// TIA Portal V18 export
// export: Created 2025-12-01T17:50:52.6792263Z, ExportSetting None, DisplayName Totally Integrated Automation Portal, DisplayVersion V18 Update 5, DisplayName TIA Portal Openness, DisplayVersion V18 Update 5, DisplayName TIA Portal Teamcenter Gateway, DisplayVersion V18, DisplayName TIA Portal Version Control Interface, DisplayVersion V18, DisplayName STEP 7 Professional, DisplayVersion V18 Update 5, DisplayName STEP 7 Safety, DisplayVersion V18, DisplayName WinCC Professional, DisplayVersion V18 Update 5
FUNCTION_BLOCK "ST10_Flow23_KReserveLifting"   // FB1093, GRAPH
// stored: AcknowledgeErrorsRequired false, AutoNumber false, GraphVersion 6.0, InitialValuesAcquisition false, SetENOAutomatically false
   // inherited from GRAPH_BASE
   VAR_INPUT
      iSysInface : "RCS_SysComInterface_V1";
   END_VAR
   VAR_IN_OUT
      ioPM_Inface : "RCS_PMInterface_V1";
      ioStatus : Int;
   END_VAR
   VAR
      sCtrlMode { S7_SetPoint := 'True'} : "SysFlowCtrlGraph";
      sUpdMES_Data : Bool;   // 更新MES数据
      工件放行中 : Bool;
      前站站号 { ExternalAccessible := 'False'; ExternalVisible := 'False'; ExternalWritable := 'False'} : UInt;
      本站站号 { ExternalAccessible := 'False'; ExternalVisible := 'False'; ExternalWritable := 'False'} : UInt;
      弹窗Temp : Array[1..10] of Int;
      AlarmID : Int;
      TON { S7_SetPoint := 'True'} : Array[0..10] of TON_TIME;
      TOF { S7_SetPoint := 'True'} : Array[0..10] of TOF_TIME;
      sUP { S7_SetPoint := 'True'} : Array[0..10] of Bool;
      更新RFID完成 : Bool;
   END_VAR
   VAR_TEMP
      Tempresult : USInt;
      本站站号乘10 : UInt;
   END_VAR
   // // TON[0] : 托盘流入1托盘到位传感器 / iA-Rotating product Check
   // // TON[1] : 托盘流入1托盘到位传感器
   // // TON[2] : 托盘流入1产品有无传感器
   // // TON[3] : 托盘流入1产品有无传感器
   // // TON[4] : 托盘流入1姿态检测光电2
   // // TON[5] : 托盘流入1姿态检测光电3
   // // TON[0].Q : 托盘流入1托盘到位 / iA-Rotating product Check
   // // TON[1].Q : 托盘流入1托盘无
   // // TON[2].Q : 托盘流入1有产品
   // // TON[3].Q : 托盘流入1无产品
   // // TON[4].Q : 托盘流入1姿态检测光电2
   // // TON[5].Q : 托盘流入1姿态检测光电3
   // // TOF[1] : iA-Rotating product Check
BEGIN
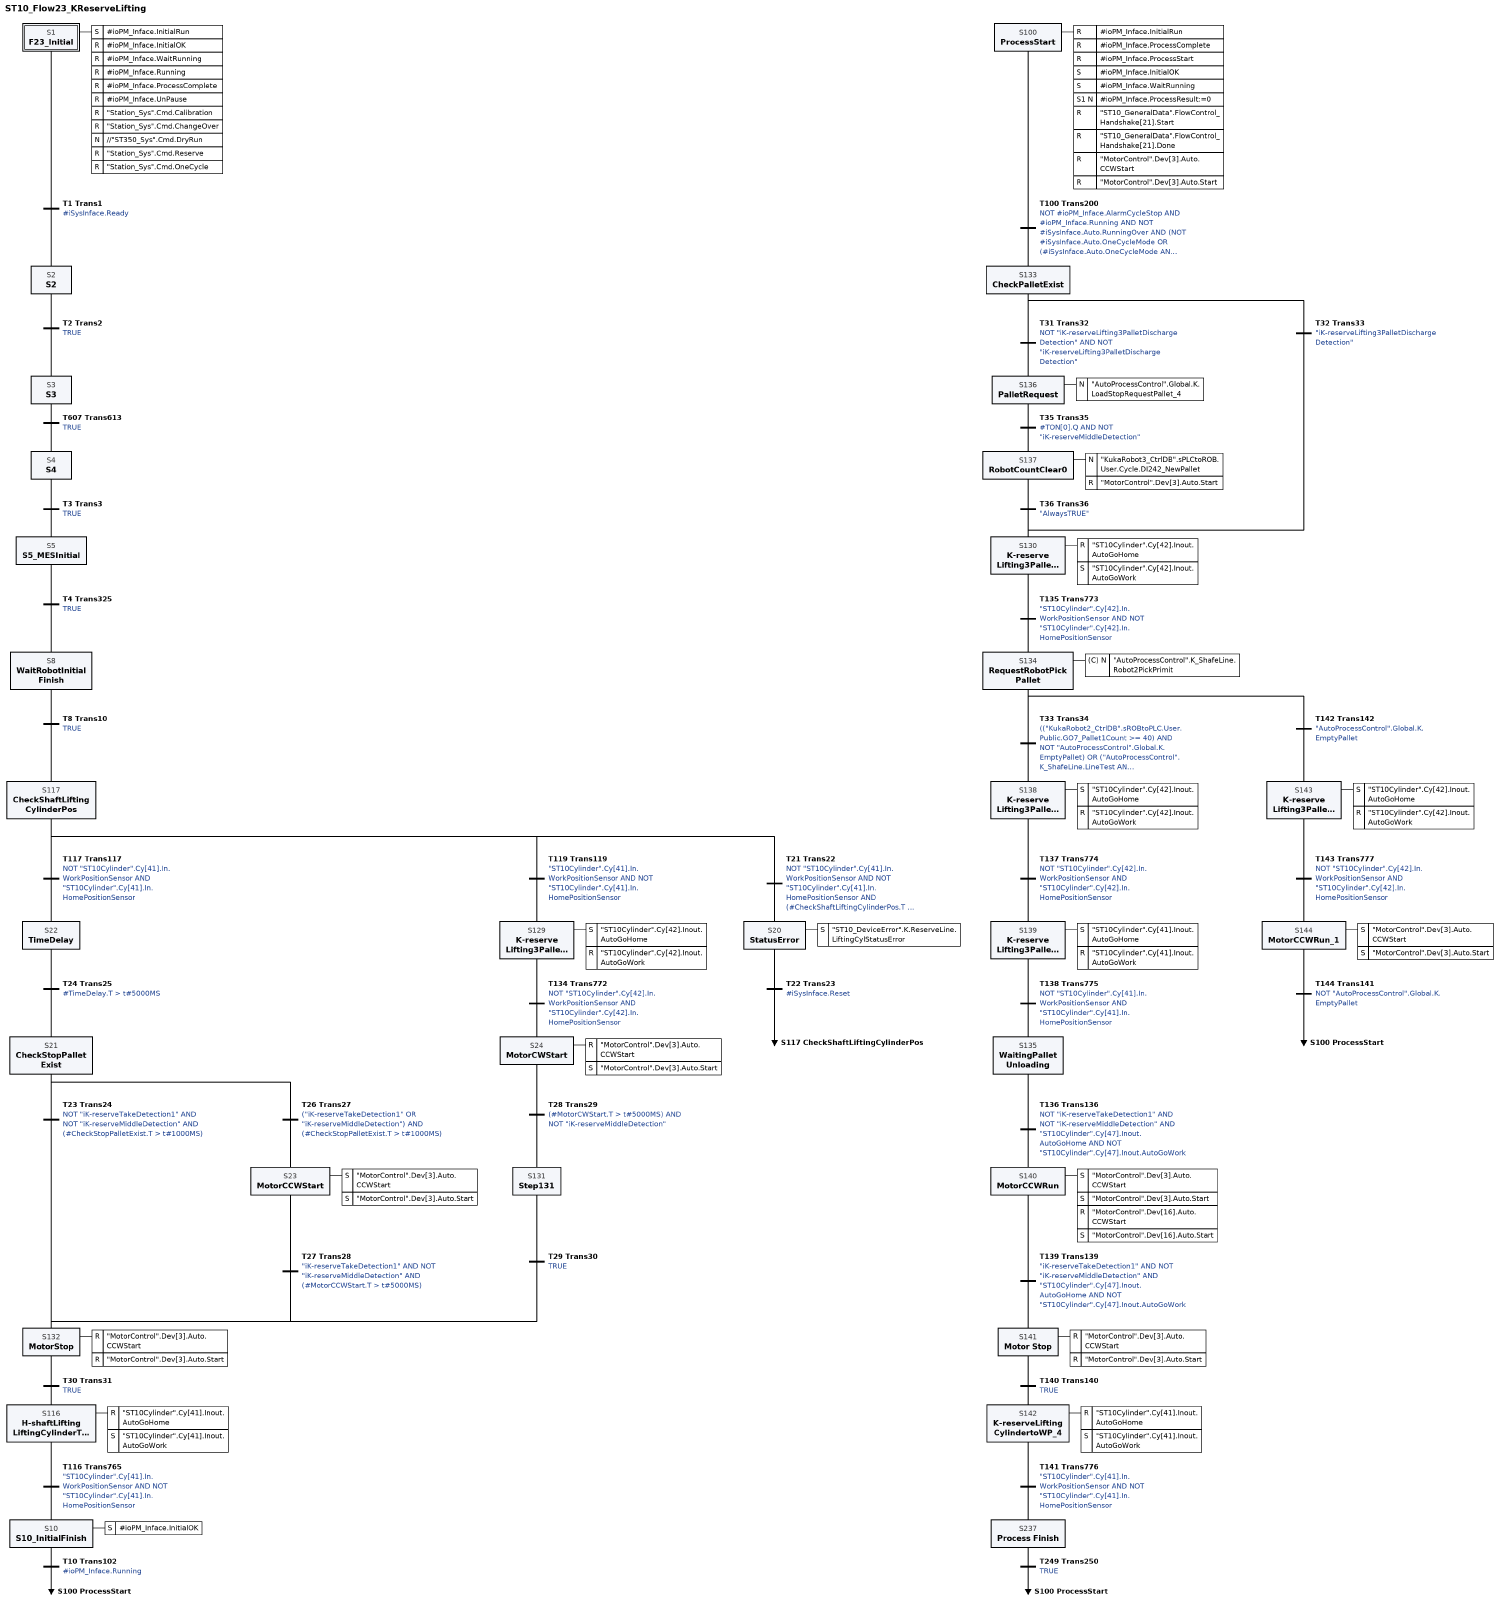
   // permanent pre-instructions
   NETWORK 1
      #TON[10].TON(IN := "AlwaysTRUE" AND "Station_Sys".Alarm.ImmediatelyStop, PT := T#300ms);
      #ioPM_Inface.AlarmImdilyStop := #TON[10].Q;
      #ioPM_Inface.AlarmCycleStop := "AlwaysTRUE" AND "Station_Sys".Alarm.CycleStop;
   NETWORK 2
      IF NOT False THEN
          #sCtrlMode(iSysInface := #iSysInface, ioPM_Inface := #ioPM_Inface, ioGraphCtrl := #RT_DATA.MOP);   // "SysFlowCtrlGraph"
      END_IF;
   NETWORK 3
      #TON[0].TON(IN := "AlwaysTRUE" AND "iK-reserveLifting3PalletDischargeDetection", PT := t#1000ms);   // 工位11有托盘
      #TOF[1].TOF(IN := "AlwaysTRUE" AND NOT "iK-reserveLifting3PalletDischargeDetection", PT := T#300ms);   // 工位无托盘
      #TON[2].TON(IN := "AlwaysTRUE", PT := T#300ms);
      #TOF[3].TOF(IN := "AlwaysTRUE", PT := T#300ms);
      #TON[4].TON(IN := "AlwaysTRUE", PT := T#300ms);
      #TOF[5].TOF(IN := "AlwaysTRUE", PT := T#300ms);
   NETWORK 4
      #前站站号 := 345;
      #本站站号 := 350;

   // sequencer 1: S01-S99 初始化 / S01-S99 Initial
   INITIAL_STEP F23_Initial:   // S1, max time T#10S, warning time T#7S
              S    #ioPM_Inface.InitialRun
              R    #ioPM_Inface.InitialOK
              R    #ioPM_Inface.WaitRunning
              R    #ioPM_Inface.Running
              R    #ioPM_Inface.ProcessComplete
              R    #ioPM_Inface.UnPause
              R    "Station_Sys".Cmd.Calibration
              R    "Station_Sys".Cmd.ChangeOver
                   //"ST350_Sys".Cmd.DryRun
              R    "Station_Sys".Cmd.Reserve
              R    "Station_Sys".Cmd.OneCycle
   END_STEP
   TRANSITION Trans1 FROM F23_Initial TO S2   // T1
      := #iSysInface.Ready;
   END_TRANSITION
   STEP S2:   // S2, max time T#10S, warning time T#7S
   END_STEP
   TRANSITION Trans2 FROM S2 TO S3   // T2
      := TRUE;
   END_TRANSITION
   STEP S4:   // S4, max time T#10S, warning time T#7S
   END_STEP
   TRANSITION Trans3 FROM S4 TO S5_MESInitial   // T3
      := TRUE;
   END_TRANSITION
   STEP S5_MESInitial:   // S5, max time T#10S, warning time T#7S
   END_STEP
   TRANSITION Trans325 FROM S5_MESInitial TO WaitRobotInitialFinish   // T4
      := TRUE;
   END_TRANSITION
   STEP S10_InitialFinish:   // S10, max time T#10S, warning time T#7S
              S    #ioPM_Inface.InitialOK
   END_STEP
   TRANSITION Trans102 FROM S10_InitialFinish TO ProcessStart   // T10, jump
      := #ioPM_Inface.Running;
   END_TRANSITION
   STEP S3:   // S3, max time T#10S, warning time T#7S
   END_STEP
   TRANSITION Trans613 FROM S3 TO S4   // T607
      := TRUE;
   END_TRANSITION
   STEP WaitRobotInitialFinish:   // S8, max time T#10S, warning time T#7S
   END_STEP
   TRANSITION Trans10 FROM WaitRobotInitialFinish TO CheckShaftLiftingCylinderPos   // T8
      := TRUE;
   END_TRANSITION
   STEP Step131:   // S131, max time T#10S, warning time T#7S
   END_STEP
   TRANSITION Trans30 FROM Step131 TO MotorStop   // T29
      := TRUE;
   END_TRANSITION
   STEP CheckShaftLiftingCylinderPos:   // S117, max time T#10S, warning time T#7S
   END_STEP
   TRANSITION Trans117 FROM CheckShaftLiftingCylinderPos TO TimeDelay   // T117
      := NOT "ST10Cylinder".Cy[41].In.WorkPositionSensor AND "ST10Cylinder".Cy[41].In.HomePositionSensor;
   END_TRANSITION
   TRANSITION Trans119 FROM CheckShaftLiftingCylinderPos TO "K-reserveLifting3PalletLocationCylindertoHP"   // T119
      := "ST10Cylinder".Cy[41].In.WorkPositionSensor AND NOT "ST10Cylinder".Cy[41].In.HomePositionSensor;
   END_TRANSITION
   TRANSITION Trans22 FROM CheckShaftLiftingCylinderPos TO StatusError   // T21
      := NOT "ST10Cylinder".Cy[41].In.WorkPositionSensor AND NOT "ST10Cylinder".Cy[41].In.HomePositionSensor AND (#CheckShaftLiftingCylinderPos.T > t#2000MS);
   END_TRANSITION
   STEP "H-shaftLiftingLiftingCylinderToWP":   // S116, max time T#10S, warning time T#7S
              R    "ST10Cylinder".Cy[41].Inout.AutoGoHome
              S    "ST10Cylinder".Cy[41].Inout.AutoGoWork
   END_STEP
   TRANSITION Trans765 FROM "H-shaftLiftingLiftingCylinderToWP" TO S10_InitialFinish   // T116
      := "ST10Cylinder".Cy[41].In.WorkPositionSensor AND NOT "ST10Cylinder".Cy[41].In.HomePositionSensor;
   END_TRANSITION
   STEP StatusError:   // S20, max time T#10S, warning time T#7S
              S    "ST10_DeviceError".K.ReserveLine.LiftingCylStatusError
   END_STEP
   TRANSITION Trans23 FROM StatusError TO CheckShaftLiftingCylinderPos   // T22, jump
      := #iSysInface.Reset;
   END_TRANSITION
   STEP CheckStopPalletExist:   // S21, max time T#10S, warning time T#7S
   END_STEP
   TRANSITION Trans24 FROM CheckStopPalletExist TO MotorStop   // T23
      := NOT "iK-reserveTakeDetection1" AND NOT "iK-reserveMiddleDetection" AND (#CheckStopPalletExist.T > t#1000MS);
   END_TRANSITION
   TRANSITION Trans27 FROM CheckStopPalletExist TO MotorCCWStart   // T26
      := ("iK-reserveTakeDetection1" OR "iK-reserveMiddleDetection") AND (#CheckStopPalletExist.T > t#1000MS);
   END_TRANSITION
   STEP TimeDelay:   // S22, max time T#10S, warning time T#7S
   END_STEP
   TRANSITION Trans25 FROM TimeDelay TO CheckStopPalletExist   // T24
      := #TimeDelay.T > t#5000MS;
   END_TRANSITION
   STEP MotorCCWStart:   // S23, max time T#10S, warning time T#7S
              S    "MotorControl".Dev[3].Auto.CCWStart
              S    "MotorControl".Dev[3].Auto.Start
   END_STEP
   TRANSITION Trans28 FROM MotorCCWStart TO MotorStop   // T27
      := "iK-reserveTakeDetection1" AND NOT "iK-reserveMiddleDetection" AND (#MotorCCWStart.T > t#5000MS);
   END_TRANSITION
   STEP MotorCWStart:   // S24, max time T#10S, warning time T#7S
              R    "MotorControl".Dev[3].Auto.CCWStart
              S    "MotorControl".Dev[3].Auto.Start
   END_STEP
   TRANSITION Trans29 FROM MotorCWStart TO Step131   // T28
      := (#MotorCWStart.T > t#5000MS) AND NOT "iK-reserveMiddleDetection";
   END_TRANSITION
   STEP "K-reserveLifting3PalletLocationCylindertoHP":   // S129, max time T#10S, warning time T#7S
              S    "ST10Cylinder".Cy[42].Inout.AutoGoHome
              R    "ST10Cylinder".Cy[42].Inout.AutoGoWork
   END_STEP
   TRANSITION Trans772 FROM "K-reserveLifting3PalletLocationCylindertoHP" TO MotorCWStart   // T134
      := NOT "ST10Cylinder".Cy[42].In.WorkPositionSensor AND "ST10Cylinder".Cy[42].In.HomePositionSensor;
   END_TRANSITION
   STEP MotorStop:   // S132, max time T#10S, warning time T#7S
              R    "MotorControl".Dev[3].Auto.CCWStart
              R    "MotorControl".Dev[3].Auto.Start
   END_STEP
   TRANSITION Trans31 FROM MotorStop TO "H-shaftLiftingLiftingCylinderToWP"   // T30
      := TRUE;
   END_TRANSITION

   // sequencer 2: S100-S199 等待到位 / S100-S199 CheckPalletStatus
   STEP ProcessStart:   // S100, max time T#10S, warning time T#7S
      // 自动等待开始运行
              R    #ioPM_Inface.InitialRun
              R    #ioPM_Inface.ProcessComplete
              R    #ioPM_Inface.ProcessStart
              S    #ioPM_Inface.InitialOK
              S    #ioPM_Inface.WaitRunning
          S1  N    #ioPM_Inface.ProcessResult:=0
              R    "ST10_GeneralData".FlowControl_Handshake[21].Start
              R    "ST10_GeneralData".FlowControl_Handshake[21].Done
              R    "MotorControl".Dev[3].Auto.CCWStart
              R    "MotorControl".Dev[3].Auto.Start
   END_STEP
   TRANSITION Trans200 FROM ProcessStart TO CheckPalletExist   // T100
      := NOT #ioPM_Inface.AlarmCycleStop AND #ioPM_Inface.Running AND NOT #iSysInface.Auto.RunningOver AND (NOT #iSysInface.Auto.OneCycleMode OR (#iSysInface.Auto.OneCycleMode AND #ioPM_Inface.TriggerOneCycle));
   END_TRANSITION
   STEP "Process Finish":   // S237, max time T#10S, warning time T#7S
   END_STEP
   TRANSITION Trans250 FROM "Process Finish" TO ProcessStart   // T249, jump
      := TRUE;
   END_TRANSITION
   STEP PalletRequest:   // S136, max time T#10S, warning time T#7S
      interlock C := NOT "Station_Sys".Cmd.ClearFlags;
              N    "AutoProcessControl".Global.K.LoadStopRequestPallet_4
   END_STEP
   TRANSITION Trans35 FROM PalletRequest TO RobotCountClear0   // T35
      := #TON[0].Q AND NOT "iK-reserveMiddleDetection";
   END_TRANSITION
   STEP WaitingPalletUnloading:   // S135, max time T#10S, warning time T#7S
   END_STEP
   TRANSITION Trans136 FROM WaitingPalletUnloading TO MotorCCWRun   // T136
      := NOT "iK-reserveTakeDetection1" AND NOT "iK-reserveMiddleDetection" AND "ST10Cylinder".Cy[47].Inout.AutoGoHome AND NOT "ST10Cylinder".Cy[47].Inout.AutoGoWork;
   END_TRANSITION
   STEP RequestRobotPickPallet:   // S134, max time T#10S, warning time T#7S
      interlock C := NOT "AutoProcessControl".Global.K.EmptyPallet AND NOT "AutoProcessControl".K_ShafeLine.LineTest;
      (C)     N    "AutoProcessControl".K_ShafeLine.Robot2PickPrimit
   END_STEP
   TRANSITION Trans34 FROM RequestRobotPickPallet TO "K-reserveLifting3PalletLocationCylindertoHP_2"   // T33
      := (("KukaRobot2_CtrlDB".sROBtoPLC.User.Public.GO7_Pallet1Count >= 40) AND NOT "AutoProcessControl".Global.K.EmptyPallet) OR ("AutoProcessControl".K_ShafeLine.LineTest AND (#RequestRobotPickPallet.T > t#2000MS));
   END_TRANSITION
   TRANSITION Trans142 FROM RequestRobotPickPallet TO "K-reserveLifting3PalletLocationCylindertoHP_4"   // T142
      := "AutoProcessControl".Global.K.EmptyPallet;
   END_TRANSITION
   STEP RobotCountClear0:   // S137, max time T#10S, warning time T#7S
              N    "KukaRobot3_CtrlDB".sPLCtoROB.User.Cycle.DI242_NewPallet
              R    "MotorControl".Dev[3].Auto.Start
   END_STEP
   TRANSITION Trans36 FROM RobotCountClear0 TO "K-reserveLifting3PalletLocationCylindertoWP_1"   // T36
      := "AlwaysTRUE";
   END_TRANSITION
   STEP CheckPalletExist:   // S133, max time T#10S, warning time T#7S
   END_STEP
   TRANSITION Trans32 FROM CheckPalletExist TO PalletRequest   // T31
      := NOT "iK-reserveLifting3PalletDischargeDetection" AND NOT "iK-reserveLifting3PalletDischargeDetection";
   END_TRANSITION
   TRANSITION Trans33 FROM CheckPalletExist TO "K-reserveLifting3PalletLocationCylindertoWP_1"   // T32
      := "iK-reserveLifting3PalletDischargeDetection";
   END_TRANSITION
   STEP "K-reserveLifting3PalletLocationCylindertoWP_1":   // S130, max time T#10S, warning time T#7S
              R    "ST10Cylinder".Cy[42].Inout.AutoGoHome
              S    "ST10Cylinder".Cy[42].Inout.AutoGoWork
   END_STEP
   TRANSITION Trans773 FROM "K-reserveLifting3PalletLocationCylindertoWP_1" TO RequestRobotPickPallet   // T135
      := "ST10Cylinder".Cy[42].In.WorkPositionSensor AND NOT "ST10Cylinder".Cy[42].In.HomePositionSensor;
   END_TRANSITION
   STEP "K-reserveLifting3PalletLocationCylindertoHP_2":   // S138, max time T#10S, warning time T#7S
              S    "ST10Cylinder".Cy[42].Inout.AutoGoHome
              R    "ST10Cylinder".Cy[42].Inout.AutoGoWork
   END_STEP
   TRANSITION Trans774 FROM "K-reserveLifting3PalletLocationCylindertoHP_2" TO "K-reserveLifting3PalletLocationCylindertoHP_3"   // T137
      := NOT "ST10Cylinder".Cy[42].In.WorkPositionSensor AND "ST10Cylinder".Cy[42].In.HomePositionSensor;
   END_TRANSITION
   STEP "K-reserveLifting3PalletLocationCylindertoHP_3":   // S139, max time T#10S, warning time T#7S
              S    "ST10Cylinder".Cy[41].Inout.AutoGoHome
              R    "ST10Cylinder".Cy[41].Inout.AutoGoWork
   END_STEP
   TRANSITION Trans775 FROM "K-reserveLifting3PalletLocationCylindertoHP_3" TO WaitingPalletUnloading   // T138
      := NOT "ST10Cylinder".Cy[41].In.WorkPositionSensor AND "ST10Cylinder".Cy[41].In.HomePositionSensor;
   END_TRANSITION
   STEP MotorCCWRun:   // S140, max time T#10S, warning time T#7S
              S    "MotorControl".Dev[3].Auto.CCWStart
              S    "MotorControl".Dev[3].Auto.Start
              R    "MotorControl".Dev[16].Auto.CCWStart
              S    "MotorControl".Dev[16].Auto.Start
   END_STEP
   TRANSITION Trans139 FROM MotorCCWRun TO "Motor Stop"   // T139
      := "iK-reserveTakeDetection1" AND NOT "iK-reserveMiddleDetection" AND "ST10Cylinder".Cy[47].Inout.AutoGoHome AND NOT "ST10Cylinder".Cy[47].Inout.AutoGoWork;
   END_TRANSITION
   STEP "Motor Stop":   // S141, max time T#10S, warning time T#7S
              R    "MotorControl".Dev[3].Auto.CCWStart
              R    "MotorControl".Dev[3].Auto.Start
   END_STEP
   TRANSITION Trans140 FROM "Motor Stop" TO "K-reserveLiftingCylindertoWP_4"   // T140
      := TRUE;
   END_TRANSITION
   STEP "K-reserveLiftingCylindertoWP_4":   // S142, max time T#10S, warning time T#7S
              R    "ST10Cylinder".Cy[41].Inout.AutoGoHome
              S    "ST10Cylinder".Cy[41].Inout.AutoGoWork
   END_STEP
   TRANSITION Trans776 FROM "K-reserveLiftingCylindertoWP_4" TO "Process Finish"   // T141
      := "ST10Cylinder".Cy[41].In.WorkPositionSensor AND NOT "ST10Cylinder".Cy[41].In.HomePositionSensor;
   END_TRANSITION
   STEP "K-reserveLifting3PalletLocationCylindertoHP_4":   // S143, max time T#10S, warning time T#7S
              S    "ST10Cylinder".Cy[42].Inout.AutoGoHome
              R    "ST10Cylinder".Cy[42].Inout.AutoGoWork
   END_STEP
   TRANSITION Trans777 FROM "K-reserveLifting3PalletLocationCylindertoHP_4" TO MotorCCWRun_1   // T143
      := NOT "ST10Cylinder".Cy[42].In.WorkPositionSensor AND "ST10Cylinder".Cy[42].In.HomePositionSensor;
   END_TRANSITION
   STEP MotorCCWRun_1:   // S144, max time T#10S, warning time T#7S
              S    "MotorControl".Dev[3].Auto.CCWStart
              S    "MotorControl".Dev[3].Auto.Start
   END_STEP
   TRANSITION Trans141 FROM MotorCCWRun_1 TO ProcessStart   // T144, jump
      := NOT "AutoProcessControl".Global.K.EmptyPallet;
   END_TRANSITION

   // permanent post-instructions
   NETWORK 1
      #ioPM_Inface.StepNum := #RT_DATA.S_DISPLAY;
   NETWORK 2
      IF #iSysInface.Reset THEN #AlarmID := 0; END_IF;
   NETWORK 3
      #TON[10].TON(IN := #工件放行中, PT := T#0.5S);
      IF #TON[10].Q THEN #工件放行中 := FALSE; END_IF;
END_FUNCTION_BLOCK
